KUKA KRL program: Fork_00_Calibration.src

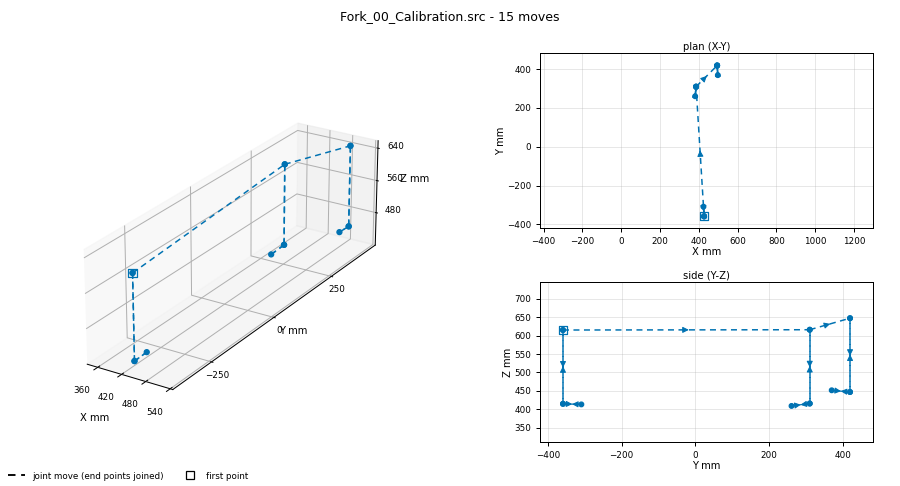
[picture p0: tool path of Fork_00_Calibration.src, 15 of 17 moves have a stored position in this frame; points joined in program order, loops and branches not executed]
&ACCESS RVP
&REL 1
&PARAM TEMPLATE = C:\KRC\Roboter\Template\vorgabe
&PARAM EDITMASK = *
DEF calibration_1 ( )


;FOLD INI
;FOLD BASISTECH INI
GLOBAL INTERRUPT DECL 3 WHEN $STOPMESS==TRUE DO IR_STOPM ( )
INTERRUPT ON 3
BAS (#INITMOV,0 )
;ENDFOLD (BASISTECH INI)
;ENDFOLD (INI)

;FOLD STARTPOSITION - BASE IS 0, TOOL IS 5, SPEED IS 15%, POSITION IS A1 5,A2 -90,A3 100,A4 5,A5 -10,A6 -5,E1 0,E2 0,E3 0,E4 0
$BWDSTART = FALSE
PDAT_ACT = {VEL 15,ACC 100,APO_DIST 50}
FDAT_ACT = {TOOL_NO 5,BASE_NO 0,IPO_FRAME #BASE}
BAS (#PTP_PARAMS,15)
PTP  {A1 5,A2 -90,A3 100,A4 5,A5 -10,A6 -5,E1 0,E2 0,E3 0,E4 0}
;ENDFOLD

;FOLD LIN SPEED IS 0.1 m/sec, INTERPOLATION SETTINGS IN FOLD
$VEL.CP=0.1
$ADVANCE=3
;ENDFOLD

BAS(#VEL_PTP,10)
PTP {X 427.493, Y -358.958, Z 615.119, A 93.883, B 1.797, C 179.999, E1 0, E2 0, E3 0, E4 0, S 'B010'} C_PTP
PTP {X 427.493, Y -358.958, Z 415.119, A 93.883, B 1.797, C 179.999, E1 0, E2 0, E3 0, E4 0, S 'B010'} C_PTP
BAS(#VEL_PTP,2)
PTP {X 424.109, Y -309.097, Z 413.551, A 93.883, B 1.797, C 179.999, E1 0, E2 0, E3 0, E4 0, S 'B010'}
BAS(#VEL_PTP,10)
PTP {X 427.493, Y -358.958, Z 415.119, A 93.883, B 1.797, C 179.999, E1 0, E2 0, E3 0, E4 0, S 'B010'} C_PTP
PTP {X 427.493, Y -358.958, Z 615.119, A 93.883, B 1.797, C 179.999, E1 0, E2 0, E3 0, E4 0, S 'B010'} C_PTP
PTP {X 386.192, Y 309.768, Z 615.9, A -95.499, B 7.507, C -90.74, E1 0, E2 0, E3 0, E4 0, S 'B010'} C_PTP
PTP {X 386.192, Y 309.768, Z 415.9, A -95.499, B 7.507, C -90.74, E1 0, E2 0, E3 0, E4 0, S 'B010'} C_PTP
BAS(#VEL_PTP,2)
PTP {X 381.441, Y 260.425, Z 409.368, A -95.499, B 7.507, C -90.74, E1 0, E2 0, E3 0, E4 0, S 'B010'}
BAS(#VEL_PTP,10)
PTP {X 386.192, Y 309.768, Z 415.9, A -95.499, B 7.507, C -90.74, E1 0, E2 0, E3 0, E4 0, S 'B010'} C_PTP
PTP {X 386.192, Y 309.768, Z 615.9, A -95.499, B 7.507, C -90.74, E1 0, E2 0, E3 0, E4 0, S 'B010'} C_PTP
PTP {X 494.791, Y 418.96, Z 647.145, A -85.926, B -5.333, C -90.376, E1 0, E2 0, E3 0, E4 0, S 'B010'} C_PTP
PTP {X 494.791, Y 418.96, Z 447.145, A -85.926, B -5.333, C -90.376, E1 0, E2 0, E3 0, E4 0, S 'B010'} C_PTP
BAS(#VEL_PTP,2)
PTP {X 498.328, Y 369.302, Z 451.793, A -85.926, B -5.333, C -90.376, E1 0, E2 0, E3 0, E4 0, S 'B010'}
BAS(#VEL_PTP,10)
PTP {X 494.791, Y 418.96, Z 447.145, A -85.926, B -5.333, C -90.376, E1 0, E2 0, E3 0, E4 0, S 'B010'} C_PTP
PTP {X 494.791, Y 418.96, Z 647.145, A -85.926, B -5.333, C -90.376, E1 0, E2 0, E3 0, E4 0, S 'B010'} C_PTP
PTP {A1 5, A2 -90, A3 100, A4 5, A5 -10, A6 -5, E1 0, E2 0, E3 0, E4 0} C_PTP

END
